FUNCTION_BLOCK Q_SoftKeyMask_AUI (* Command change soft key mask with AUI adapter ( Part 6 - F.36 ) *)
  (* Standard: ISO 11783-6; Description: Copyright (c) 2026 Meisterschulen am Ostbahnhof This program and the accompanying materials are made available under the terms of the Eclipse Public License 2.0 which is available at https://www.eclipse.org/legal/epl-2.0/ SPDX-License-Identifier: EPL-2.0 *)
  (* Version 1.0, 2026-09-11, Franz Höpfinger, Meisterschulen am Ostbahnhof, AUI adapter wrapper for Q_SoftKeyMask *)
  PACKAGE isobus::UT::Q;
  IMPORT isobus::UT::Q::const::IDs::ID_NULL;
  (* Documentation:
  Command change soft key mask with AUI adapter ( Part 6 - F.36 )
   This FB is an AUI adapter wrapper around Q_SoftKeyMask.
  *)
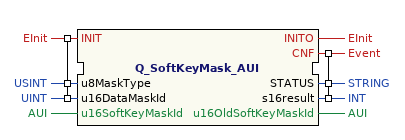
  EVENT_INPUT
    INIT : EInit WITH u8MaskType, u16DataMaskId; (* Service Initialization *)
  END_EVENT
  EVENT_OUTPUT
    INITO : EInit; (* Initialization Confirm *)
    CNF WITH STATUS, s16result; (* Confirmation of Requested Service *)
  END_EVENT
  VAR_INPUT
    u8MaskType : USINT; (* Mask Type (1: DataMask, 2: AlarmMask) *)
    u16DataMaskId : UINT := ID_NULL; (* Object ID of data/alarm mask *)
  END_VAR
  VAR_OUTPUT
    STATUS : STRING; (* Service Status *)
    s16result : INT; (* retval see description *)
  END_VAR
  SOCKETS
    u16SoftKeyMaskId : adapter::types::unidirectional::AUI; (* New soft key mask ID *)
  END_SOCKETS
  PLUGS
    u16OldSoftKeyMaskId : adapter::types::unidirectional::AUI; (* Old soft key mask ID *)
  END_PLUGS
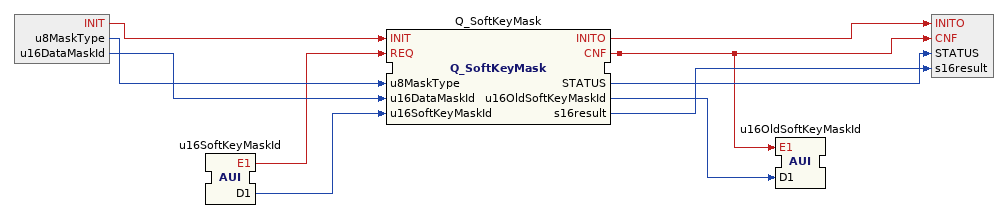
  FBS
    Q_SoftKeyMask : isobus::UT::Q::Q_SoftKeyMask;
  END_FBS
  EVENT_CONNECTIONS
    INIT TO Q_SoftKeyMask.INIT;
    Q_SoftKeyMask.INITO TO INITO;
    Q_SoftKeyMask.CNF TO CNF;
    u16SoftKeyMaskId.E1 TO Q_SoftKeyMask.REQ;
    Q_SoftKeyMask.CNF TO u16OldSoftKeyMaskId.E1;
  END_CONNECTIONS
  DATA_CONNECTIONS
    Q_SoftKeyMask.STATUS TO STATUS;
    u8MaskType TO Q_SoftKeyMask.u8MaskType;
    u16DataMaskId TO Q_SoftKeyMask.u16DataMaskId;
    u16SoftKeyMaskId.D1 TO Q_SoftKeyMask.u16SoftKeyMaskId;
    Q_SoftKeyMask.u16OldSoftKeyMaskId TO u16OldSoftKeyMaskId.D1;
    Q_SoftKeyMask.s16result TO s16result;
  END_CONNECTIONS
END_FUNCTION_BLOCK
